// TIA Portal V17 export
// export: Created 2025-06-26T06:33:56.8111617Z, ExportSetting WithDefaults, DisplayName Totally Integrated Automation Portal, DisplayVersion V17 Update 8, DisplayName TIA Portal Openness, DisplayVersion V17 Update 8, DisplayName TIA Portal Version Control Interface, DisplayVersion V17, DisplayName STEP 7 Professional, DisplayVersion V17 Update 8, DisplayName STEP 7 Safety, DisplayVersion V17 Update 6, DisplayName WinCC Advanced, DisplayVersion V17 Update 8
FUNCTION "isNaN" : Bool   // FC19, FBD
TITLE = isNaN
{ S7_Optimized_Access := 'TRUE' }
VERSION : 0.1
// Returns TRUE if a REAL is NaN
// stored: AutoNumber true, IsIECCheckEnabled false, SetENOAutomatically false, UDAEnableTagReadback false
   VAR_INPUT
      In : Real;
   END_VAR
BEGIN

REGION Network 1
   // NOT_OK is a compiler builtin, but not available in SCL
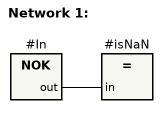
   // no SCL statement known for NOK: written as a call
   #isNaN := NOK(#In);
END_REGION
END_FUNCTION
